INTERFACE I_Insertion2D

METHOD ABSTRACT align : BOOL
VAR_INPUT
	targetPos : REAL;
END_VAR
END_METHOD

PROPERTY Busy : BOOL
GET
END_GET
SET
END_SET
END_PROPERTY

PROPERTY Contact : BOOL
GET
END_GET
SET
END_SET
END_PROPERTY

PROPERTY Home : BOOL
GET
END_GET
SET
END_SET
END_PROPERTY

METHOD ABSTRACT homingSequence : BOOL
VAR_INPUT
END_VAR
END_METHOD

METHOD ABSTRACT press : BOOL
VAR_INPUT
END_VAR
END_METHOD

METHOD ABSTRACT release : BOOL
VAR_INPUT
END_VAR
END_METHOD

PROPERTY ScrewPos : LREAL
GET
END_GET
SET
END_SET
END_PROPERTY

PROPERTY SliderPos : LREAL
GET
END_GET
SET
END_SET
END_PROPERTY

METHOD ABSTRACT traverse : BOOL
VAR_INPUT
	direction : MC_Direction;
END_VAR
END_METHOD

END_INTERFACE

(* stored: Version 1.1.0.1, ProductVersion 3.1.4024.11
   Itf I_Insertion2D: Id {8e64ce60-22e0-4b91-ba46-fa91d2f7ae0e}
   Folder Properties: Id {4db86ba3-5e15-4610-89d6-3573b1563320}
   Method align: Id {fa643266-3d8f-4e66-aec5-e5710590bff8}
   Property Busy: Id {22835791-0cba-4766-a640-8df2ffdb894d}
   Get Get: Id {c91d3a80-05fd-4fd9-93ce-86b32db3d06b}
   Set Set: Id {f282b493-143e-481d-a756-b09c263b633b}
   Property Contact: Id {88516ae2-b7cf-49c6-8562-f4f20559cb97}
   Get Get: Id {b65e7839-b08d-41e0-b5f3-e57ba70a0f47}
   Set Set: Id {4df19e98-4f82-40e8-8c7a-f9016f0511fc}
   Property Home: Id {2e214f8e-025e-4655-8dbf-fc929a398aaf}
   Get Get: Id {6f3cd418-c02e-46d8-a44d-e21e27ce2eb6}
   Set Set: Id {7506060e-75ba-48f2-803d-dc66f4e7419f}
   Method homingSequence: Id {e50d8f3c-3832-479d-9ea8-d077b3535f03}
   Method press: Id {d84955f1-e0a2-4a22-92a7-c7477ef94736}
   Method release: Id {92bdeeca-e13f-4d7f-bf24-c4aad1f47945}
   Property ScrewPos: Id {0f9296b0-dac0-4298-8710-e435017a1512}
   Get Get: Id {f4c321d6-5acd-437d-ae12-0a22a0a9b2c4}
   Set Set: Id {bcb2ca56-e8a3-4b99-b659-d2adaedd2baf}
   Property SliderPos: Id {a384a15a-0431-4fb8-ad53-2f38f4c7c81a}
   Get Get: Id {6754d911-f109-4572-b856-7f898a9cd456}
   Set Set: Id {ac2b81d2-5a59-463d-8eb5-09c8cf0faf42}
   Method traverse: Id {62c2b24a-3291-4b2f-ac0b-b5af5509b392} *)
